{attribute addProperty BoxType "EL3773-0000-0018"}
{attribute addProperty Id "U2_StatusAT %I*U2_Status_E2EFACF1162"}
{attribute addProperty CRC "4034060072"}
{attribute addProperty SizeInBites "16"}
{attribute addProperty SizeInBytes "2"}
TYPE L2_Voltage_Status_F072DF28 :
STRUCT
	{attribute addProperty Name "U2_Status"}
	U2_Status AT %I* : U2_Status_E2EFACF1;
END_STRUCT
END_TYPE

(* stored: Version 1.2.0.0, ProductVersion 3.1.4024.9
   DUT L2_Voltage_Status_F072DF28: Id {abe7e601-f371-427c-af10-37dd40047467} *)
